(* CODESYS project OkayToBag.xml

Project tree, tasks and I/O mapping:
  function OkayToBag [LD]
*)

// OkayToBag
FUNCTION OkayToBag : BOOL
// Function to check if all components are ready to make a bag of ice.
VAR_INPUT
	BagCount:			BOOL;				//
	BagPresent:			BOOL;				//
	DoorLocked:			BOOL;				//
	IceLevel:			BOOL;				//
	HeatSeal:			BOOL;				//
	Heater:				BOOL;				//
	Kicker:				BOOL;				//
END_VAR
VAR
END_VAR

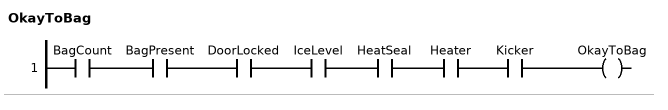
// NETWORK 1
OkayToBag := BagCount AND BagPresent AND DoorLocked AND IceLevel AND HeatSeal AND Heater AND Kicker;

END_FUNCTION
